(* Schneider Machine Expert - Basic project water_pump_realpars_video, file version 2.7.0.0 *)
(* ProjectInformations: Name=New project *)

HARDWARE
  Cpu 0: TM221M16R/G
  EthernetConfiguration: NetworkName=M221, IpAllocationMode=FixedAddress, IpAddress=0.0.0.0, SubnetMask=0.0.0.0
  SerialLineConfiguration: Baud=Baud19200, Parity=ParityEven, DataBits=DataBits8, StopBits=StopBits1, PhysicalMedium=PhysicalMediumRs485, TransmissionMode=TransmissionModeModbusRtu, SlaveId=1, Addressing=SlaveAddressing
  MastTask: UsePeriodScanMode=false, PeriodScan=100
  FastTask: Period=255
  CpuBehavior: StartingMode=StartAsPreviousState, AutoSaveRamOnEeprom=true, WatchdogPeriod=250

SYMBOLS  (address, symbol, comment, settings)
  %TM0        [Used=true, Type=TOF, Preset=7, Base=OneSecond]
  %I0.0     STARTED
  %I0.1     LLS
  %I0.2     HLS
  %I0.3     STOP
  %Q0.0     PUMP1
  %Q0.1     PUMP2
  %Q0.2     MIXER
  %Q0.3     VALVE

GRAFCET Grafcet POU
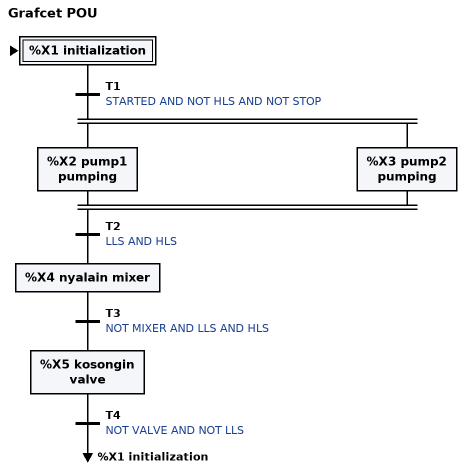
  INITIAL_STEP %X1  (* initialization *)
  STEP %X2  (* pump1 pumping *)
  STEP %X3  (* pump2 pumping *)
  STEP %X4  (* nyalain mixer *)
  STEP %X5  (* kosongin valve *)
  TRANSITION T1 FROM %X1 TO %X2, %X3 := STARTED AND NOT HLS AND NOT STOP;
  TRANSITION T2 FROM %X2, %X3 TO %X4 := LLS AND HLS;
  TRANSITION T3 FROM %X4 TO %X5 := NOT MIXER AND LLS AND HLS;
  TRANSITION T4 FROM %X5 TO %X1 := NOT VALVE AND NOT LLS;

STEP %X2 pump1 pumping
  (* SectionNumber=2, StepNumber=2 *)

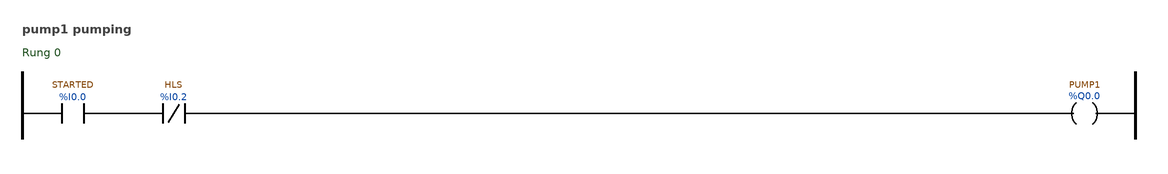

// Rung 0
  LD %I0.0                (* STARTED *)
  ANDN %I0.2              (* HLS *)
  ST %Q0.0                (* PUMP1 *)
  // as ST:
  //   PUMP1 := STARTED AND NOT HLS;

TRANSITION T1 (%X1 -> %X2, %X3) 
  (* SectionNumber=0 *)

// Rung 1: tombol start ditekan
  LD %I0.0                (* STARTED *)
  ANDN %I0.2              (* HLS *)
  ANDN %I0.3              (* STOP *)
  ENDT
  // as ST:
  //   TRANSITION := STARTED AND NOT HLS AND NOT STOP;

STEP %X3 pump2 pumping
  (* SectionNumber=3, StepNumber=3 *)

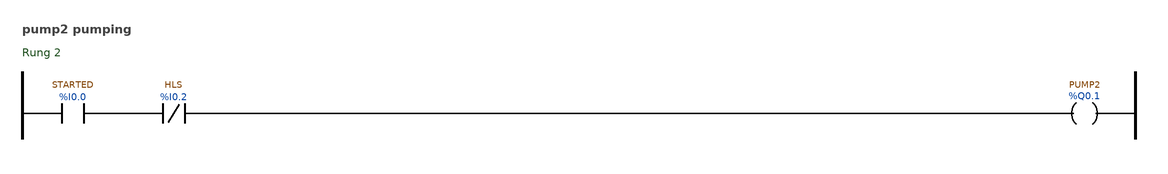

// Rung 2
  LD %I0.0                (* STARTED *)
  ANDN %I0.2              (* HLS *)
  ST %Q0.1                (* PUMP2 *)
  // as ST:
  //   PUMP2 := STARTED AND NOT HLS;

STEP %X4 nyalain mixer
  (* SectionNumber=4, StepNumber=4 *)

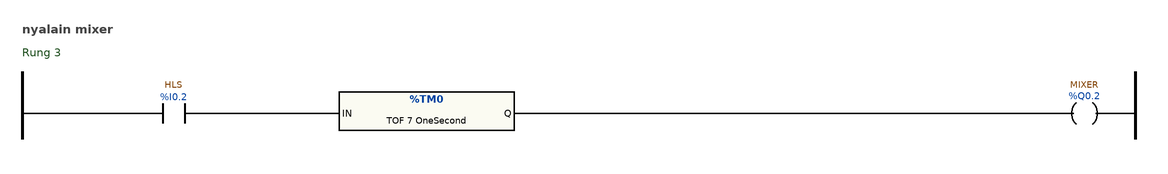

// Rung 3
  BLK %TM0
  LD %I0.2                (* HLS *)
  IN
  OUT_BLK
  LD Q
  ST %Q0.2                (* MIXER *)
  END_BLK
  // as ST:
  //   %TM0(IN := HLS);
  //   MIXER := %TM0.Q;

STEP %X5 kosongin valve
  (* SectionNumber=5, StepNumber=5 *)

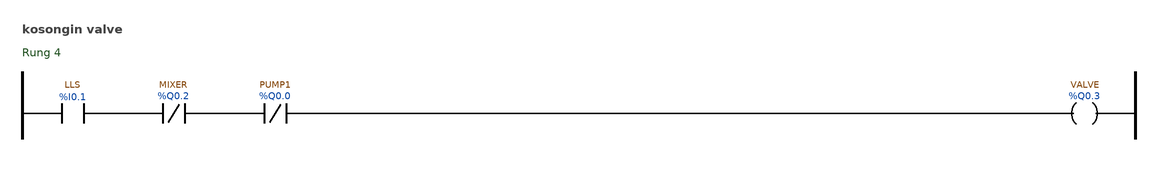

// Rung 4
  LD %I0.1                (* LLS *)
  ANDN %Q0.2              (* MIXER *)
  ANDN %Q0.0              (* PUMP1 *)
  ST %Q0.3                (* VALVE *)
  // as ST:
  //   VALVE := LLS AND NOT MIXER AND NOT PUMP1;

TRANSITION T2 (%X2, %X3 -> %X4) 
  (* SectionNumber=0 *)

// Rung 5: ls1
  LD %I0.1                (* LLS *)
  AND %I0.2               (* HLS *)
  ENDT
  // as ST:
  //   TRANSITION := LLS AND HLS;

TRANSITION T3 (%X4 -> %X5) 
  (* SectionNumber=0 *)

// Rung 6: WAIT 7S
  LDN %Q0.2               (* MIXER *)
  AND %I0.1               (* LLS *)
  AND %I0.2               (* HLS *)
  ENDT
  // as ST:
  //   TRANSITION := NOT MIXER AND LLS AND HLS;

TRANSITION T4 (%X5 -> %X1) 
  (* SectionNumber=0 *)

// Rung 7: PROSES COMPLETED
  LDN %Q0.3               (* VALVE *)
  ANDN %I0.1              (* LLS *)
  ENDT
  // as ST:
  //   TRANSITION := NOT VALVE AND NOT LLS;
